FUNCTION_BLOCK Linearachse
VAR_INPUT
END_VAR
VAR_OUTPUT
END_VAR
VAR
END_VAR

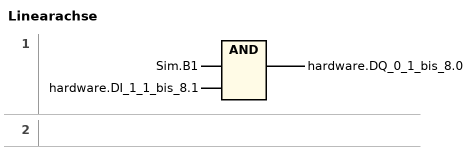
// NETWORK 1
hardware.DQ_0_1_bis_8.0 := Sim.B1 AND hardware.DI_1_1_bis_8.1;

// NETWORK 2

END_FUNCTION_BLOCK

(* stored: Version 1.1.0.1, ProductVersion 3.1.4024.5
   POU Linearachse: Id {3114a163-c196-4be2-ab35-6259f5e7c1b4}, SpecialFunc None *)
